PROGRAM MAIN
VAR
END_VAR

END_PROGRAM

(* stored: Version 1.1.0.1
   POU MAIN: Id {5c7536fb-b230-4ec9-a902-58b9d7780b0e} *)
